FUNCTION_BLOCK adapterTest (* Composite Function Block Type *)
  (* Standard: 61499-2 *)
  (* Version 0.0, 2014-04-02, 4DIAC-IDE, 4DIAC-Consortium *)
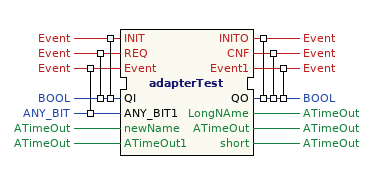
  EVENT_INPUT
    INIT WITH QI; (* Initialization Request *)
    REQ WITH QI; (* Normal Execution Request *)
    Event WITH ANY_BIT1;
  END_EVENT
  EVENT_OUTPUT
    INITO WITH QO; (* Initialization Confirm *)
    CNF WITH QO; (* Execution Confirmation *)
    Event1 WITH QO;
  END_EVENT
  VAR_INPUT
    QI : BOOL; (* Input event qualifier *)
    ANY_BIT1 : ANY_BIT;
  END_VAR
  VAR_OUTPUT
    QO : BOOL; (* Output event qualifier *)
  END_VAR
  SOCKETS
    newName : ATimeOut;
    ATimeOut1 : ATimeOut;
  END_SOCKETS
  PLUGS
    LongNAme : ATimeOut;
    ATimeOut : ATimeOut;
    short : ATimeOut;
  END_PLUGS
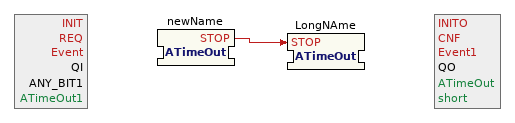
  EVENT_CONNECTIONS
    newName.STOP TO LongNAme.STOP;
  END_CONNECTIONS
END_FUNCTION_BLOCK
